FUNCTION_BLOCK DoorController (* Basic Function Block Type *)
  (* Standard: 61499-2 *)
  (* Version 0.0, 9/24/2026, macie, Schneider Electric, Template *)
  PACKAGE Main;
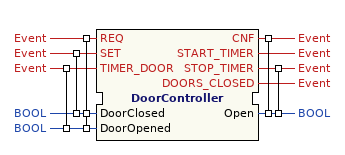
  EVENT_INPUT
    REQ WITH DoorClosed, DoorOpened; (* Normal Execution Request *)
    SET WITH DoorClosed;
    TIMER_DOOR WITH DoorOpened;
  END_EVENT
  EVENT_OUTPUT
    CNF WITH Open; (* Execution Confirmation *)
    START_TIMER;
    STOP_TIMER WITH Open;
    DOORS_CLOSED;
  END_EVENT
  VAR_INPUT
    DoorClosed : BOOL;
    DoorOpened : BOOL;
  END_VAR
  VAR_OUTPUT
    Open : BOOL; (* Output event qualifier *)
  END_VAR
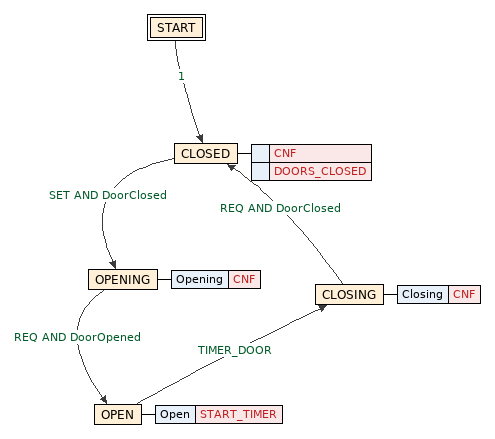
  EC_STATES
    START; (* Initial State *)
    CLOSED : -> CNF, -> DOORS_CLOSED;
    OPENING : Opening -> CNF;
    OPEN : Open -> START_TIMER;
    CLOSING : Closing -> CNF;
  END_STATES
  EC_TRANSITIONS
    START TO CLOSED := 1;
    CLOSED TO OPENING := SET AND DoorClosed;
    OPENING TO OPEN := REQ AND DoorOpened;
    OPEN TO CLOSING := TIMER_DOOR;
    CLOSING TO CLOSED := REQ AND DoorClosed;
  END_TRANSITIONS
  ALGORITHM Opening IN ST: (* Initialization algorithm *)
;
Open := TRUE;
  END_ALGORITHM
  ALGORITHM Closing IN ST:
;
Open := FALSE;
  END_ALGORITHM
  ALGORITHM Open IN ST:
;
  END_ALGORITHM
END_FUNCTION_BLOCK
